// TIA Portal V17 export
// export: Created 2022-04-29T00:39:00.3711304Z, ExportSetting WithDefaults, DisplayName Totally Integrated Automation Portal, DisplayVersion V17, DisplayName TIA Portal Openness, DisplayVersion V17, DisplayName TIA Portal Version Control Interface, DisplayVersion V17, DisplayName STEP 7 Professional, DisplayVersion V17, DisplayName STEP 7 Safety, DisplayVersion V17, DisplayName WinCC Advanced, DisplayVersion V17
FUNCTION "Multiply" : Void   // FC1, LAD
{ S7_Optimized_Access := 'TRUE' }
VERSION : 0.1
// stored: AutoNumber true, IsIECCheckEnabled false, SetENOAutomatically false, UDAEnableTagReadback false
   VAR_INPUT
      In1 : Real;
      In2 : Real;
   END_VAR
   VAR_OUTPUT
      Out : Real;
   END_VAR
BEGIN

REGION Network 1: Multiply
   // This is a simple comment
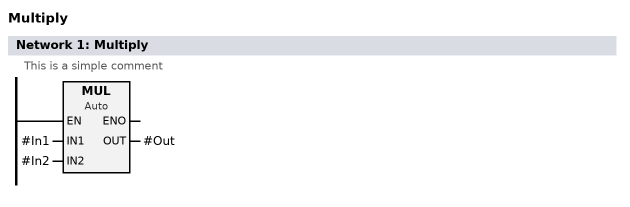
   RUNG wire#powerrail
      Mul(in1 := #In1, in2 := #In2, out => #Out)
   END_RUNG
   // the same network as SCL:
   #Out := #In1 * #In2;
END_REGION
END_FUNCTION
